INTERFACE I_Shape

METHOD M_Draw : BOOL
VAR_INPUT
END_VAR
END_METHOD

END_INTERFACE

(* stored: Version 1.1.0.1, ProductVersion 3.1.4024.12
   Itf I_Shape: Id {b631e55d-f627-4300-9f17-b03966c3422d}
   Method M_Draw: Id {fa87e993-e59e-40a5-bd81-7731214f8dae} *)
